(* CoDeSys 2.3 export: PARALISTENTRY_TS.EXP *)

(* Data type in Diag/Other *)
TYPE ParaListEntry_ts :
STRUCT
	Description_as8		: STRING(32);
(*	Description_as8		: ARRAY [1..4] OF STRING(32);*)
END_STRUCT
END_TYPE
